(* Logix 5000 project; controller Empty vendor 1 type 14 code 226 rev 34.11; software revision 34.01 *)

TASK Fast (periodic, rate 100 ms, priority 1, watchdog 150 ms) : FastProgram
TASK loop (continuous, watchdog 1000 ms) : MainProgram
TASK Normal (periodic, rate 250 ms, priority 2, watchdog 375 ms) : NormalProgram
TASK SafetyTask (periodic, rate 20 ms, priority 10, watchdog 20 ms, safety) : SafetyProgram
TASK Slow (periodic, rate 500 ms, priority 3, watchdog 750 ms) : SlowProgram
TASK System (periodic, rate 1000 ms, priority 4, watchdog 1500 ms) : SystemProgram

MODULES
   Local : vendor 1 type 14 code 226 (5069 0, rev 34.11)
END_MODULES

PROGRAM FastProgram   (* main routine MainRoutine *)

ROUTINE MainRoutine   (* ladder *)
END_ROUTINE
END_PROGRAM

PROGRAM MainProgram   (* main routine main *)
VAR
   counter : LINT;
END_VAR

ROUTINE main   (* structured text *)
   
   
   counter := 100_000;
   
   WHILE counter >= 0 DO
   	counter := counter - 1;
   END_WHILE;
   
   
   
   
END_ROUTINE
END_PROGRAM

PROGRAM NormalProgram   (* main routine MainRoutine *)

ROUTINE MainRoutine   (* ladder *)
END_ROUTINE
END_PROGRAM

PROGRAM SafetyProgram   (* main routine MainRoutine, safety *)

ROUTINE MainRoutine   (* ladder *)
END_ROUTINE
END_PROGRAM

PROGRAM SlowProgram   (* main routine MainRoutine *)

ROUTINE MainRoutine   (* ladder *)
END_ROUTINE
END_PROGRAM

PROGRAM SystemProgram   (* main routine MainRoutine *)

ROUTINE MainRoutine   (* ladder *)
END_ROUTINE
END_PROGRAM
